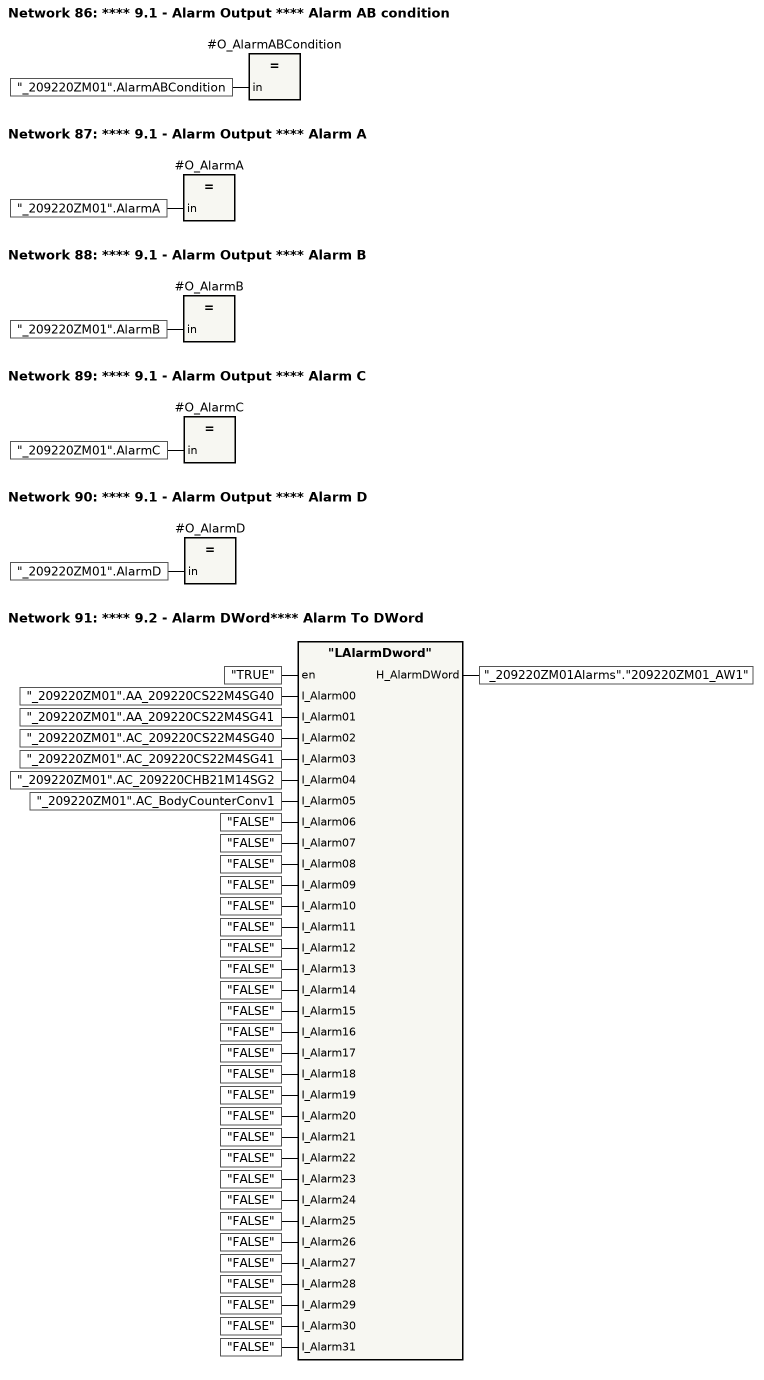
   #O_AlarmABCondition := "_209220ZM01".AlarmABCondition;
END_REGION

REGION Network 87: **** 9.1 - Alarm Output **** Alarm A
   // Output Alarm A
   #O_AlarmA := "_209220ZM01".AlarmA;
END_REGION

REGION Network 88: **** 9.1 - Alarm Output **** Alarm B
   // Output Alarm B
   #O_AlarmB := "_209220ZM01".AlarmB;
END_REGION

REGION Network 89: **** 9.1 - Alarm Output **** Alarm C
   // Output Alarm A
   #O_AlarmC := "_209220ZM01".AlarmC;
END_REGION

REGION Network 90: **** 9.1 - Alarm Output **** Alarm D
   // Output Alarm D
   #O_AlarmD := "_209220ZM01".AlarmD;
END_REGION

REGION Network 91: **** 9.2 - Alarm DWord**** Alarm To DWord
   // Alarm Word
   IF "TRUE" THEN
       "LAlarmDword"(I_Alarm00 := "_209220ZM01".AA_209220CS22M4SG40,
                     I_Alarm01 := "_209220ZM01".AA_209220CS22M4SG41,
                     I_Alarm02 := "_209220ZM01".AC_209220CS22M4SG40,
                     I_Alarm03 := "_209220ZM01".AC_209220CS22M4SG41,
                     I_Alarm04 := "_209220ZM01".AC_209220CHB21M14SG2,
                     I_Alarm05 := "_209220ZM01".AC_BodyCounterConv1,
                     I_Alarm06 := "FALSE",
                     I_Alarm07 := "FALSE",
                     I_Alarm08 := "FALSE",
                     I_Alarm09 := "FALSE",
                     I_Alarm10 := "FALSE",
                     I_Alarm11 := "FALSE",
                     I_Alarm12 := "FALSE",
                     I_Alarm13 := "FALSE",
                     I_Alarm14 := "FALSE",
                     I_Alarm15 := "FALSE",
                     I_Alarm16 := "FALSE",
                     I_Alarm17 := "FALSE",
                     I_Alarm18 := "FALSE",
                     I_Alarm19 := "FALSE",
                     I_Alarm20 := "FALSE",
                     I_Alarm21 := "FALSE",
                     I_Alarm22 := "FALSE",
                     I_Alarm23 := "FALSE",
                     I_Alarm24 := "FALSE",
                     I_Alarm25 := "FALSE",
                     I_Alarm26 := "FALSE",
                     I_Alarm27 := "FALSE",
                     I_Alarm28 := "FALSE",
                     I_Alarm29 := "FALSE",
                     I_Alarm30 := "FALSE",
                     I_Alarm31 := "FALSE",
                     H_AlarmDWord => "_209220ZM01Alarms"."209220ZM01_AW1");
   END_IF;
END_REGION
END_FUNCTION
